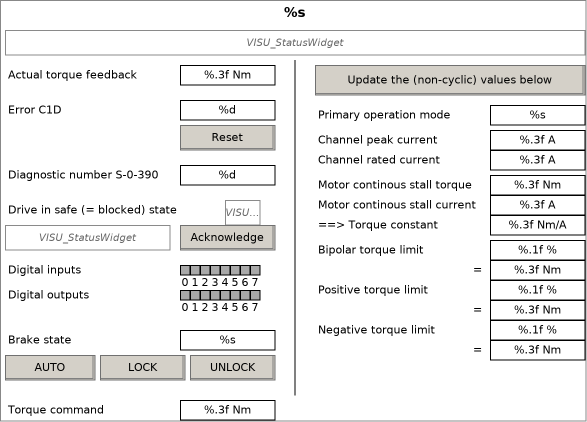
VISUALIZATION VISU_AX522DriveChannel  // 587x422
VAR_IN_OUT
    ref : AX52XXDriveChannel;
    widget : AX52XXDriveChannelWidget;
END_VAR
    Frame (5,30 580x25)
        shows VISU_StatusWidget(widget := widget.actualStatus)
    Rectangle (5,0 580x25), "%s", text variable: widget.name
    Label (315,130 175x20), "Channel peak current"
    Rectangle (490,130 95x20), "%.3f A", text variable: ref.channelPeakCurrent.amps.value
    Label (315,150 175x20), "Channel rated current"
    Rectangle (490,150 95x20), "%.3f A", text variable: ref.channelRatedCurrent.amps.value
    Label (315,175 175x20), "Motor continous stall torque"
    Label (315,195 175x20), "Motor continous stall current"
    Rectangle (490,175 95x20), "%.3f Nm", text variable: ref.continuousStallTorque.newtonmeter.value
    Rectangle (490,195 95x20), "%.3f A", text variable: ref.continuousStallCurrent.amps.value
    Label (315,215 175x20), "==> Torque constant"
    Rectangle (490,215 95x20), "%.3f Nm/A", text variable: ref.torqueConstant
    Button (315,65 270x30), "Update the (non-cyclic) values below", input disabled if: ref.processes.update.statuses.enabledStatus.disabled
        OnMouseClick: execute { ref.processes.update.do_request := TRUE; }
    Label (315,240 175x20), "Bipolar torque limit"
    Rectangle (490,240 95x20), "%.1f %", text variable: ref.bipolarTorqueLimit.percent.value
    Rectangle (490,260 95x20), "%.3f Nm", text variable: ref.bipolarTorqueLimit.newtonmeter.value
    Label (470,260 20x20), "="
    Label (315,280 175x20), "Positive torque limit"
    Rectangle (490,280 95x20), "%.1f %", text variable: ref.positiveTorqueLimit.percent.value
    Rectangle (490,300 95x20), "%.3f Nm", text variable: ref.positiveTorqueLimit.newtonmeter.value
    Label (470,300 20x20), "="
    Label (315,320 175x20), "Negative torque limit"
    Rectangle (490,320 95x20), "%.1f %", text variable: ref.negativeTorqueLimit.percent.value
    Rectangle (490,340 95x20), "%.3f Nm", text variable: ref.negativeTorqueLimit.newtonmeter.value
    Label (470,340 20x20), "="
    Label (5,65 175x20), "Actual torque feedback"
    Rectangle (180,65 95x20), "%.3f Nm", text variable: ref.actualTorqueFeedback.newtonmeter.value
    Label (5,100 175x20), "Error C1D"
    Rectangle (180,100 95x20), "%d", text variable: ref.errorC1D
    Label (5,260 175x20), "Digital inputs"
    Rectangle (180,265 10x10), colour toggle: widget.input0
    Label (180,275 10x15), "0"
    Label (190,275 10x15), "1"
    Label (200,275 10x15), "2"
    Label (210,275 10x15), "3"
    Label (220,275 10x15), "4"
    Label (230,275 10x15), "5"
    Label (240,275 10x15), "6"
    Label (250,275 10x15), "7"
    Rectangle (190,265 10x10), colour toggle: widget.input1
    Rectangle (200,265 10x10), colour toggle: widget.input2
    Rectangle (210,265 10x10), colour toggle: widget.input3
    Rectangle (220,265 10x10), colour toggle: widget.input4
    Rectangle (230,265 10x10), colour toggle: widget.input5
    Rectangle (240,265 10x10), colour toggle: widget.input6
    Rectangle (250,265 10x10), colour toggle: widget.input7
    Label (5,285 175x20), "Digital outputs"
    Rectangle (180,290 10x10), colour toggle: widget.output0
    Label (180,300 10x15), "0"
    Label (190,300 10x15), "1"
    Label (200,300 10x15), "2"
    Label (210,300 10x15), "3"
    Label (220,300 10x15), "4"
    Label (230,300 10x15), "5"
    Label (240,300 10x15), "6"
    Label (250,300 10x15), "7"
    Rectangle (190,290 10x10), colour toggle: widget.output1
    Rectangle (200,290 10x10), colour toggle: widget.output2
    Rectangle (210,290 10x10), colour toggle: widget.output3
    Rectangle (220,290 10x10), colour toggle: widget.output4
    Rectangle (230,290 10x10), colour toggle: widget.output5
    Rectangle (240,290 10x10), colour toggle: widget.output6
    Rectangle (250,290 10x10), colour toggle: widget.output7
    Label (315,105 175x20), "Primary operation mode"
    Rectangle (490,105 95x20), "%s", text variable: ref.operatingMode
    Rectangle (180,330 95x20), "%s", text variable: ref.brakeState
    Label (5,330 175x20), "Brake state"
    Button (5,355 90x25), "AUTO", input disabled if: ref.processes.setBrake.statuses.enabledStatus.disabled
        OnMouseClick: execute { ref.processes.setBrake.set.newState := DriveBrakeStates.BRAKE_AUTOMATIC; ref.processes.setBrake.do_request := TRUE; }
    Button (100,355 85x25), "LOCK", input disabled if: ref.processes.setBrake.statuses.enabledStatus.disabled
        OnMouseClick: execute { ref.processes.setBrake.set.newState := DriveBrakeStates.BRAKE_FORCE_LOCK; ref.processes.setBrake.do_request := TRUE; }
    Button (190,355 85x25), "UNLOCK", input disabled if: ref.processes.setBrake.statuses.enabledStatus.disabled
        OnMouseClick: execute { ref.processes.setBrake.set.newState := DriveBrakeStates.BRAKE_FORCE_UNLOCK; ref.processes.setBrake.do_request := TRUE; }
    Line (295,395) (295,60)
    Button (180,125 95x25), "Reset", input disabled if: ref.processes.reset.statuses.enabledStatus.disabled
        OnMouseClick: execute { ref.processes.reset.do_request := TRUE; }
    Label (5,400 175x20), "Torque command", invisible if: ref.operatingMode <> DriveOperatingModes.OPERATING_MODE_TORQUE_CONTROL
    Rectangle (180,400 95x20), "%.3f Nm", text variable: ref.torqueCommand.newtonmeter.value, invisible if: ref.operatingMode <> DriveOperatingModes.OPERATING_MODE_TORQUE_CONTROL
    Label (5,165 175x20), "Diagnostic number S-0-390"
    Rectangle (180,165 95x20), "%d", text variable: ref.diagnosticNumber
    Label (5,200 215x20), "Drive in safe (= blocked) state"
    Frame (225,200 35x25)
        shows VISU_State_gray_red(state := ref.isInSafetate)
    Button (180,225 95x25), "Acknowledge", input disabled if: ref.processes.acknowledgeSafetyError.statuses.enabledStatus.disabled
        OnMouseClick: execute { ref.processes.acknowledgeSafetyError.do_request := TRUE; }
    Frame (5,225 165x25)
        shows VISU_StatusWidget(widget := widget.processes_acknowledgeSafetyError)
END_VISUALIZATION

(* stored: Version 1.1.0.1, ProductVersion 3.1.4019.2
   Visu VISU_AX522DriveChannel: Id {00d6b398-b2a8-48a2-b46f-1f6ffba431cd} *)
